// TIA Portal V18 export
FUNCTION "AHU_UnitState" : Void   // FC60100, FBD
{ S7_Optimized_Access := 'TRUE' }
VERSION : 0.1
// stored: AutoNumber false, IsIECCheckEnabled false, SetENOAutomatically false, UDAEnableTagReadback false
   VAR_INPUT
      iUnitID : Int;   // 1=AHUFood, 2=AHUNonFood
   END_VAR
   VAR_TEMP
      FA_temp : Real;
   END_VAR
BEGIN

REGION Network 1 (SCL)
   IF "FirstScan" THEN
       ;
       "AHUUnitStates".UnitStates.cActual[#iUnitID] := 0;
       "AHUUnitStates".UnitStates.cTarget[#iUnitID] := 0;
   END_IF;
END_REGION

REGION Network 2: AHUs Actual Operation Mode define
   // Operation Modes                                                 Unit State
   // 0=Protection                                                         0=Stopped
   // 1=Economy                                                           1=Checking-up  
   // 2=PreComfort                                                       2=Preheating
   // 3=Comfor                                                              3=Starting 
   // 4=Auto(Scheduler)                                              4=RecirculatingOperation (Protection)
   //                                                                                 5=Sustained Mode (Economy setpoints)
   //                                                                                 6=Sustained Mode (PreComfort setpoints) 
   //                                                                                 7=Comfort  operation
   //                                                                                 8=Stopping
   //                                                                                 9=Blocking
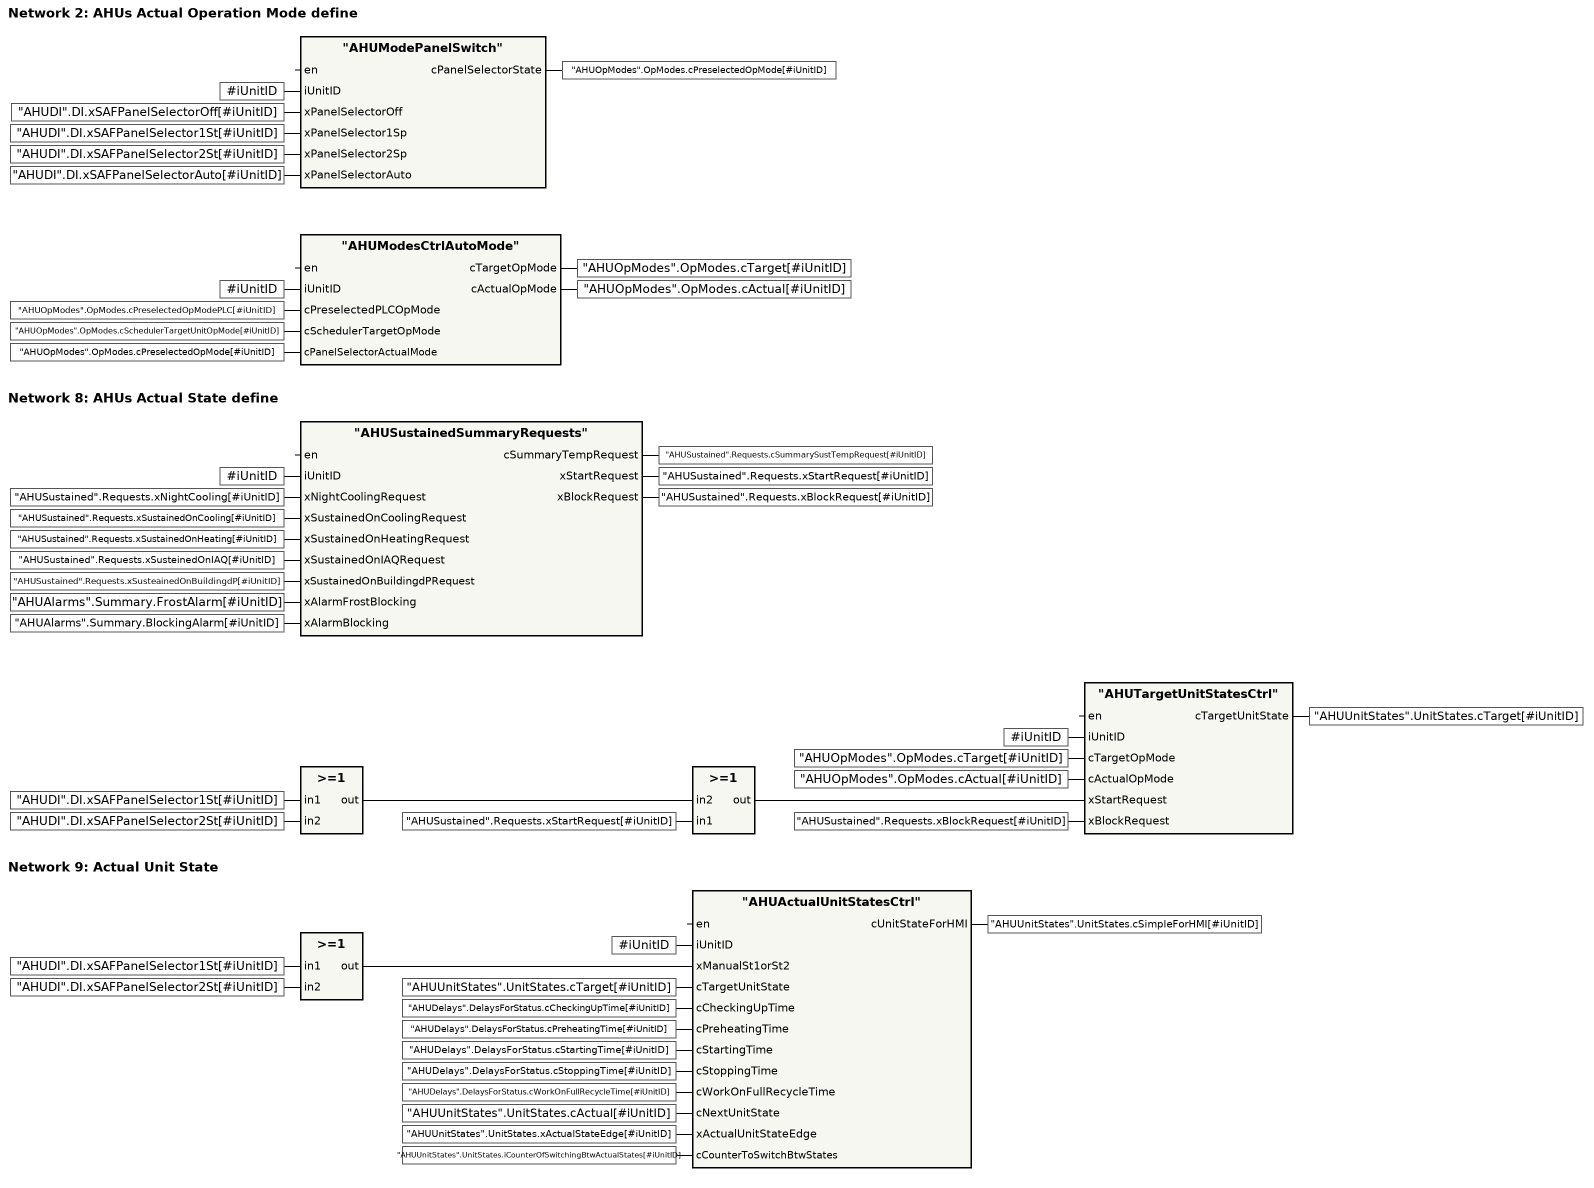
   "AHUModePanelSwitch"(iUnitID := #iUnitID,
                        xPanelSelectorOff := "AHUDI".DI.xSAFPanelSelectorOff[#iUnitID],
                        xPanelSelector1Sp := "AHUDI".DI.xSAFPanelSelector1St[#iUnitID],
                        xPanelSelector2Sp := "AHUDI".DI.xSAFPanelSelector2St[#iUnitID],
                        xPanelSelectorAuto := "AHUDI".DI.xSAFPanelSelectorAuto[#iUnitID],
                        cPanelSelectorState => "AHUOpModes".OpModes.cPreselectedOpMode[#iUnitID]);
   "AHUModesCtrlAutoMode"(iUnitID := #iUnitID,
                          cPreselectedPLCOpMode := "AHUOpModes".OpModes.cPreselectedOpModePLC[#iUnitID],
                          cSchedulerTargetOpMode := "AHUOpModes".OpModes.cSchedulerTargetUnitOpMode[#iUnitID],
                          cPanelSelectorActualMode := "AHUOpModes".OpModes.cPreselectedOpMode[#iUnitID],
                          cTargetOpMode => "AHUOpModes".OpModes.cTarget[#iUnitID],
                          cActualOpMode => "AHUOpModes".OpModes.cActual[#iUnitID]);
END_REGION

REGION Network 3 (SCL): NightCooling Request
   IF FALSE THEN
       // Statement section IF
       "AHUSustained".Requests.xNightCooling[#iUnitID] := TRUE;
   ELSE
       "AHUSustained".Requests.xNightCooling[#iUnitID] := FALSE;
   END_IF;
END_REGION

REGION Network 4 (SCL): Sustained requests cooling
   IF "AHURegulators".Regulators.State.cTempCooling[#iUnitID] > 0 THEN
       // Statement section IF
       ;
   ELSE
       "AHUSustained".Requests.xSustainedOnCooling[#iUnitID] := FALSE;
   END_IF;
END_REGION

REGION Network 5 (SCL): Sustained request heating
   IF "AHURegulators".Regulators.State.cTempHeating[#iUnitID] > 0 THEN
       // Statement section IF
       ;
   ELSE
       "AHUSustained".Requests.xSustainedOnHeating[#iUnitID] := FALSE;
   END_IF;
END_REGION

REGION Network 6 (SCL): Sustained request IAQ
   IF "AHURegulators".Regulators.State.cIAQ[#iUnitID] > 0 THEN
       // Statement section IF
       ;
   ELSE
       "AHUSustained".Requests.xSusteinedOnIAQ[#iUnitID] := FALSE;
   END_IF;
END_REGION

REGION Network 7 (SCL): Sustained request Building Pressurisation
   IF "AHURegulators".Regulators.State.cBuildingdP[#iUnitID] > 0 THEN
       // Statement section IF
       ;
   ELSE
       "AHUSustained".Requests.xSusteainedOnBuildingdP[#iUnitID] := FALSE;
   END_IF;
END_REGION

REGION Network 8: AHUs Actual State define
   // Operation Modes                                                 Unit State
   // 0=Protection                                                         0=Stopped
   // 1=Economy                                                           1=Checking-up  
   // 2=PreComfort                                                       2=Preheating
   // 3=Comfor                                                              3=Starting 
   // 4=Auto(Scheduler)                                              4=RecirculatingOperation
   //                                                                                 5=Sustained Mode (Economy setpoints)
   //                                                                                 6=Sustained Mode (PreComfort setpoints) 
   //                                                                                 7=Comfort  operation
   //                                                                                 8=Stopping
   //                                                                                 9=Blocking
   "AHUSustainedSummaryRequests"(iUnitID := #iUnitID,
                           xNightCoolingRequest := "AHUSustained".Requests.xNightCooling[#iUnitID],
                           xSustainedOnCoolingRequest := "AHUSustained".Requests.xSustainedOnCooling[#iUnitID],
                           xSustainedOnHeatingRequest := "AHUSustained".Requests.xSustainedOnHeating[#iUnitID],
                           xSustainedOnIAQRequest := "AHUSustained".Requests.xSusteinedOnIAQ[#iUnitID],
                           xSustainedOnBuildingdPRequest := "AHUSustained".Requests.xSusteainedOnBuildingdP[#iUnitID],
                           xAlarmFrostBlocking := "AHUAlarms".Summary.FrostAlarm[#iUnitID],
                           xAlarmBlocking := "AHUAlarms".Summary.BlockingAlarm[#iUnitID],
                           cSummaryTempRequest => "AHUSustained".Requests.cSummarySustTempRequest[#iUnitID],
                           xStartRequest => "AHUSustained".Requests.xStartRequest[#iUnitID],
                           xBlockRequest => "AHUSustained".Requests.xBlockRequest[#iUnitID]);
   "AHUTargetUnitStatesCtrl"(iUnitID := #iUnitID,
                           cTargetOpMode := "AHUOpModes".OpModes.cTarget[#iUnitID],
                           cActualOpMode := "AHUOpModes".OpModes.cActual[#iUnitID],
                           xStartRequest := "AHUDI".DI.xSAFPanelSelector1St[#iUnitID] OR "AHUDI".DI.xSAFPanelSelector2St[#iUnitID] OR "AHUSustained".Requests.xStartRequest[#iUnitID],
                           xBlockRequest := "AHUSustained".Requests.xBlockRequest[#iUnitID],
                           cTargetUnitState => "AHUUnitStates".UnitStates.cTarget[#iUnitID]);
END_REGION

REGION Network 9: Actual Unit State
   "AHUActualUnitStatesCtrl"(iUnitID := #iUnitID,
                           xManualSt1orSt2 := "AHUDI".DI.xSAFPanelSelector1St[#iUnitID] OR "AHUDI".DI.xSAFPanelSelector2St[#iUnitID],
                           cTargetUnitState := "AHUUnitStates".UnitStates.cTarget[#iUnitID],
                           cCheckingUpTime := "AHUDelays".DelaysForStatus.cCheckingUpTime[#iUnitID],
                           cPreheatingTime := "AHUDelays".DelaysForStatus.cPreheatingTime[#iUnitID],
                           cStartingTime := "AHUDelays".DelaysForStatus.cStartingTime[#iUnitID],
                           cStoppingTime := "AHUDelays".DelaysForStatus.cStoppingTime[#iUnitID],
                           cWorkOnFullRecycleTime := "AHUDelays".DelaysForStatus.cWorkOnFullRecycleTime[#iUnitID],
                           cNextUnitState := "AHUUnitStates".UnitStates.cActual[#iUnitID],
                           xActualUnitStateEdge := "AHUUnitStates".UnitStates.xActualStateEdge[#iUnitID],
                           cCounterToSwitchBtwStates := "AHUUnitStates".UnitStates.iCounterOfSwitchingBtwActualStates[#iUnitID],
                           cUnitStateForHMI => "AHUUnitStates".UnitStates.cSimpleForHMI[#iUnitID]);
END_REGION
END_FUNCTION
